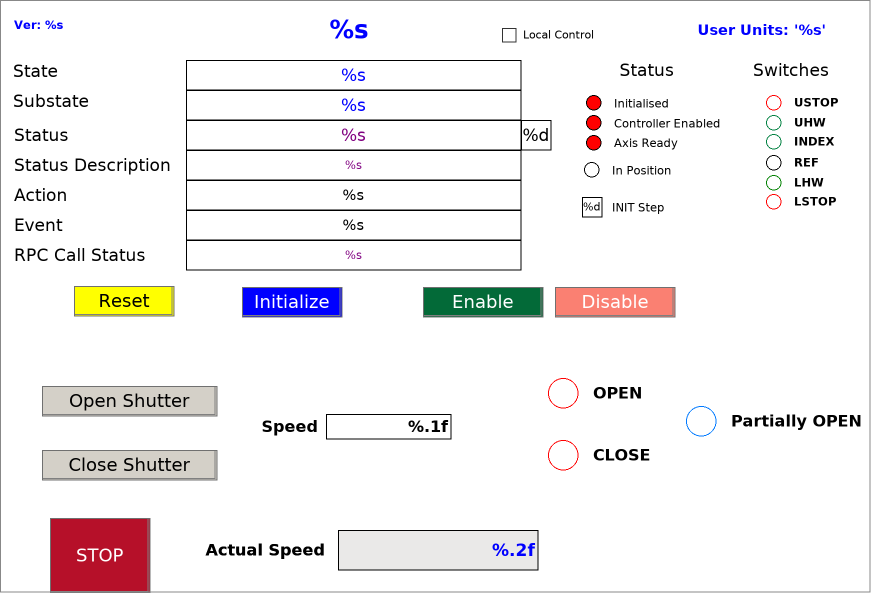
VISUALIZATION GUI_NOTT_SHUTTERS  // 871x593
    Rectangle (186,60 335x30), "%s", text variable: m_Instance.stat.sState
    Rectangle (186,90 335x30), "%s", text variable: m_Instance.stat.sSubstate
    Button (74,286 100x30), "Reset", input disabled if: NOT m_Instance.stat.bLocal OR NOT m_Instance.in_bSafe
        OnMouseDown: execute {
            m_Instance.ctrl.bLocalCmd := TRUE;
            m_Instance.ctrl.nCommand := E_MOTOR_COMMAND.RESET;
            m_Instance.ctrl.bExecute := TRUE;
        }
    Button (242,287 100x30), "Initialize", input disabled if: NOT m_Instance.stat.bLocal OR NOT m_Instance.in_bSafe
        OnMouseDown: execute {
            m_Instance.ctrl.bLocalCmd := TRUE;
            m_Instance.ctrl.nCommand := E_MOTOR_COMMAND.INIT;
            m_Instance.ctrl.bExecute := TRUE;
        }
    Button (50,518 100x75), "STOP", input disabled if: NOT m_Instance.stat.bLocal OR NOT m_Instance.in_bSafe
        OnMouseDown: execute {
            m_Instance.ctrl.bLocalCmd := TRUE;
            m_Instance.ctrl.nCommand := E_MOTOR_COMMAND.STOP;
            m_Instance.ctrl.bExecute := TRUE;
        }
    Button (423,287 120x30), "Enable", input disabled if: NOT m_Instance.stat.bLocal OR NOT m_Instance.in_bSafe
        OnMouseDown: execute {
            m_Instance.ctrl.bLocalCmd := TRUE;
            m_Instance.ctrl.nCommand := E_MOTOR_COMMAND.ENABLE;
            m_Instance.ctrl.bExecute := TRUE;
        }
    Button (555,287 120x30), "Disable", input disabled if: NOT m_Instance.stat.bLocal OR NOT m_Instance.in_bSafe
        OnMouseDown: execute {
            m_Instance.ctrl.bLocalCmd := TRUE;
            m_Instance.ctrl.nCommand := E_MOTOR_COMMAND.DISABLE;
            m_Instance.ctrl.bExecute := TRUE;
        }
    Rectangle (10,56 170x30), "State"
    Rectangle (10,86 170x30), "Substate"
    Rectangle (186,120 335x30), "%s", text variable: m_Instance.stat.sStatus
    Rectangle (186,150 335x30), "%s", tooltip "Additional information mostly used for description of errors", text variable: m_Instance.stat.sErrorText
    Rectangle (11,120 170x30), "Status"
    Rectangle (11,150 170x30), "Status Description"
    Rectangle (186,180 335x30), "%s", text variable: m_Instance.stat.sActionDesc
    Rectangle (186,210 335x30), "%s", text variable: m_Instance.stat.sEventDesc
    Rectangle (11,180 170x30), "Action"
    Rectangle (11,210 170x30), "Event"
    Rectangle (233,12 232x35), "%s", text variable: m_Instance.sName
    Checkbox (500,20 116x30), "Local Control", variable: m_Instance.stat.bLocal
    Rectangle (601,55 92x30), "Status"
    Rectangle (521,120 30x30), "%d", text variable: m_Instance.stat.nStatus
    Rectangle (745,55 92x30), "Switches"
    Rectangle (791,95 50x15), "USTOP"
    Ellipse (766,95 15x15), colour toggle: m_Instance.stat.signals[5].bActive
    Ellipse (766,115 15x15), colour toggle: m_Instance.stat.signals[4].bActive
    Ellipse (766,175 15x15), colour toggle: m_Instance.stat.signals[1].bActive
    Ellipse (766,194 15x15), colour toggle: m_Instance.stat.signals[0].bActive
    Ellipse (766,155 15x15), colour toggle: m_Instance.stat.signals[2].bActive
    Rectangle (791,134 50x15), "INDEX"
    Rectangle (791,115 50x15), "UHW"
    Rectangle (791,155 50x15), "REF"
    Rectangle (791,175 50x15), "LHW"
    Rectangle (791,194 50x15), "LSTOP"
    Ellipse (766,134 15x15), colour toggle: m_Instance.stat.signals[3].bActive
    Ellipse (586,95 15x15), tooltip "GREEN = Initialised RED = Not Initialised", text variable: m_Instance.stat.bInitialised, colour toggle: m_Instance.stat.bInitialised
    Rectangle (611,91 90x25), "Initialised"
    Rectangle (611,111 125x25), "Controller Enabled"
    Rectangle (611,131 90x24), "Axis Ready"
    Ellipse (586,115 15x15), tooltip "GREEN = Enabled RED = Disabled", colour toggle: m_Instance.stat.bEnabled
    Ellipse (586,135 15x15), tooltip "GREEN = Ready RED = Not Ready", colour toggle: m_Instance.stat.bAxisReady
    Rectangle (582,197 20x20), "%d", text variable: m_Instance.stat.nInitStep
    Rectangle (609,195 90x25), "INIT Step"
    Rectangle (11,240 170x30), "RPC Call Status"
    Rectangle (186,240 335x30), "%s", text variable: m_Instance.stat.sRPCErrorText
    Rectangle (609,158 90x25), "In Position"
    Ellipse (584,162 15x15), tooltip "GREEN = In Position BLANK = Not In Position (or not used)", colour toggle: (m_Instance.stat.bInPosition) <> 0
    Rectangle (626,15 203x30), "User Units: '%s'", text variable: m_Instance.stat.axis.sUnits
    Rectangle (11,10 99x30), "Ver: %s", tooltip "'Motor.library version'", text variable: m_Instance.stat.sLibVersion, input disabled if: true
    Group (178,530 360x40)
        Rectangle (160,0 200x40), "%.2f", text variable: m_Instance.stat.lrVelActual, input disabled if: false
        Rectangle (0,5 150x30), "Actual Speed"
    Rectangle (338,530 200x40), "%.2f", text variable: m_Instance.stat.lrVelActual, input disabled if: false
    Rectangle (178,535 150x30), "Actual Speed"
    Rectangle (226,414 95x25), "Speed", tooltip "Shutter Speed (mm/sec)"
    Rectangle (326,414 125x25), "%.1f", text variable: m_Instance.ctrl.lrVelocity
        OnMouseDown: write the text variable via Default
    Button (42,386 175x30), "Open Shutter", input disabled if: NOT m_Instance.stat.bLocal OR NOT m_Instance.in_bSafe
        OnMouseDown: execute {
            m_Instance.ctrl.bLocalCmd := TRUE;
            m_Instance.ctrl.nCommand := E_MOTOR_COMMAND.MOTOR_MOVE;
            m_Instance.ctrl.nMoveType := E_MOTOR_MOVE_TYPE.VELOCITY;
            m_Instance.ctrl.nDirection := MC_Negative_Direction;
            m_Instance.ctrl.bExecute := TRUE;
        }
    Button (42,450 175x30), "Close Shutter", input disabled if: NOT m_Instance.stat.bLocal OR NOT m_Instance.in_bSafe
        OnMouseDown: execute {
            m_Instance.ctrl.bLocalCmd := TRUE;
            m_Instance.ctrl.nCommand := E_MOTOR_COMMAND.MOTOR_MOVE;
            m_Instance.ctrl.nMoveType := E_MOTOR_MOVE_TYPE.VELOCITY;
            m_Instance.ctrl.nDirection := MC_Positive_Direction;
            m_Instance.ctrl.bExecute := TRUE;
        }
    Ellipse (548,378 30x30), colour toggle: m_Instance.stat.signals[5].bActive
    Rectangle (590,378 100x30), "OPEN", tooltip "Shutter is Open"
    Ellipse (548,440 30x30), colour toggle: m_Instance.stat.signals[0].bActive
    Rectangle (590,440 100x30), "CLOSE", tooltip "Shutter is closed"
    Ellipse (686,406 30x30), colour toggle: m_Instance.bShutterPartiallyOpen
    Rectangle (728,406 143x30), "Partially OPEN", tooltip "Either shutter is opening or closing"
END_VISUALIZATION

(* stored: Version 1.1.0.1, ProductVersion 3.1.4024.14
   Visu GUI_NOTT_SHUTTERS: Id {5e594847-9f26-4c58-8ba6-71576b082866} *)
